FUNCTION_BLOCK PML_Method_Sample EXTENDS PML_Method_Base
VAR_INPUT
END_VAR
VAR_OUTPUT
END_VAR
VAR
END_VAR

SUPER^();

END_FUNCTION_BLOCK

(* stored: Version 1.1.0.1, ProductVersion 3.1.4024.11
   POU PML_Method_Sample: Id {7017d611-2e36-4a7a-a774-9234147f3ede}, SpecialFunc None *)
